Universal Robots PolyScope program: pourAndPutDown.urp

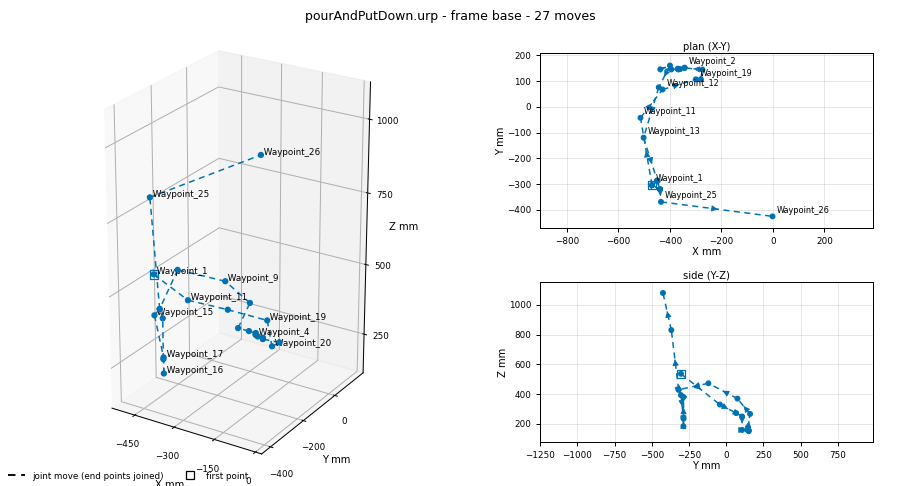
[picture p0: tool path of pourAndPutDown.urp in frame base, 27 of 27 moves have a stored position in this frame; points joined in program order, loops and branches not executed]
Program pourAndPutDown (installation=default directory=/programs/PrakjoyShi_Beer createdIn=5.12.6.1102099 lastSavedIn=5.12.6.1102099 robotSerialNumber=20215500597)
Calibrated DH parameters: a=[0.000193, -0.066673, -0.391568, -0.000012, 0.00005, 0]; d=[0.162643, -472.05677, 465.132521, 7.058239, 0.099746, 0.099582]; alpha=[1.571116, 0.00089, 0.003862, 1.569269, -1.569248, 0]; deltaTheta=[0, -1.413394, 7.628392, 0.068187, 0, -0.000001]
Robot Program (runOnlyOnce=true)
  MoveJ speed 60 deg/s, acceleration 80 deg/s^2 (useActiveTCP=true) feature=Base
    Waypoint Waypoint_1: TCP in base x=-469.422 y=-303.772 z=537.049 mm, rx=-0.9663 ry=-1.499 rz=1.6747 rad; joints [6.908, -106.662, 129.097, -206.194, -67.737, 6.591] deg; TCP offset x=0 y=0 z=191.5 mm, rx=0 ry=0 rz=0 rad
    Waypoint Waypoint_11: TCP in base x=-514.044 y=-42.229 z=330.478 mm, rx=0.9483 ry=1.8098 rz=-1.8406 rad; joints [-42.944, -57.453, 101.188, -230.29, 31.853, 49.611] deg
    Waypoint Waypoint_12: TCP in base x=-428.386 y=67.501 z=272.98 mm, rx=0.8234 ry=1.7173 rz=-1.638 rad; joints [-53.416, -47.466, 95.297, -230.558, 54.247, 53.558] deg
    Waypoint Waypoint_19: TCP in base x=-299.055 y=107.007 z=250.481 mm, rx=0.7818 ry=1.7818 rz=-1.7132 rad; joints [-69.052, -50.894, 107.804, -239.624, 68.324, 47.588] deg
    Waypoint Waypoint_20: TCP in base x=-279.734 y=106.984 z=159.803 mm, rx=0.7816 ry=1.7818 rz=-1.7132 rad; joints [-71.245, -40.233, 108.371, -250.83, 70.508, 47.507] deg
    Waypoint Waypoint_21: TCP in base x=-273.429 y=144.767 z=159.8 mm, rx=0.7817 ry=1.7819 rz=-1.7133 rad; joints [-73.337, -38.608, 103.329, -247.386, 72.596, 47.386] deg; TCP offset x=0 y=0 z=191.5 mm, rx=0 ry=0 rz=0 rad
    Waypoint Waypoint_2: TCP in base x=-342.426 y=151.266 z=151.388 mm, rx=0.9523 ry=1.6137 rz=-1.4653 rad; joints [-64.863, -34.688, 92.564, -242.174, 67.302, 65.082] deg; TCP offset x=0 y=0 z=191.5 mm, rx=0 ry=0 rz=0 rad
    Waypoint Waypoint_22: TCP in base x=-343.072 y=152.365 z=156.122 mm, rx=0.9896 ry=1.5509 rz=-1.4276 rad; joints [-64.858, -34.701, 92.594, -241.206, 67.284, 68.699] deg
    Waypoint Waypoint_3: TCP in base x=-360.092 y=146.777 z=158.442 mm, rx=1.1766 ry=1.3384 rz=-1.269 rad; joints [-64.056, -34.823, 92.755, -240.944, 64.321, 84.128] deg
    Wait Sleep waitTime=5
    Waypoint Waypoint_4: TCP in base x=-368.401 y=147.927 z=162.208 mm, rx=1.2276 ry=1.2595 rz=-1.2399 rad; joints [-64.055, -34.823, 92.749, -240.156, 62.793, 88.217] deg
    Wait Sleep waitTime=10
    Waypoint Waypoint_27: TCP in base x=-368.415 y=147.907 z=162.228 mm, rx=1.2493 ry=1.2256 rz=-1.2076 rad; joints [-64.053, -34.824, 92.753, -240.154, 62.79, 90.783] deg
    Wait Sleep waitTime=2
    Waypoint Waypoint_5: TCP in base x=-367.114 y=145.876 z=165.681 mm, rx=1.0874 ry=1.5479 rz=-1.4306 rad; joints [-64.058, -36.96, 92.743, -241.765, 62.844, 71.518] deg
    Waypoint Waypoint_6: TCP in base x=-367.053 y=145.733 z=170.165 mm, rx=0.9649 ry=1.707 rz=-1.5493 rad; joints [-64.058, -37.901, 92.741, -241.83, 62.842, 60.713] deg
    Waypoint Waypoint_7: TCP in base x=-394.155 y=145.769 z=170.181 mm, rx=0.9649 ry=1.707 rz=-1.5494 rad; joints [-61.586, -36.44, 89.13, -239.83, 60.388, 61.045] deg
    Waypoint Waypoint_8: TCP in base x=-437.191 y=145.775 z=170.185 mm, rx=0.9649 ry=1.707 rz=-1.5494 rad; joints [-57.925, -33.834, 82.842, -236.41, 56.767, 61.573] deg
    Waypoint Waypoint_10: TCP in base x=-399.525 y=160.604 z=267.522 mm, rx=0.291 ry=1.9476 rz=-1.9017 rad; joints [-57.921, -39.735, 82.866, -222.692, 65.755, 24.515] deg
    Waypoint Waypoint_9: TCP in base x=-443.299 y=75.819 z=370.314 mm, rx=-0.1462 ry=2.1698 rz=-2.071 rad; joints [-49.086, -50.8, 82.87, -214.951, 58.642, 3.159] deg
    Waypoint Waypoint_13: TCP in base x=-501.996 y=-119.391 z=473.346 mm, rx=-0.1865 ry=2.1452 rz=-2.0717 rad; joints [-29.839, -60.518, 82.876, -205.008, 41.125, 3.179] deg
    Waypoint Waypoint_14: TCP in base x=-438.339 y=-319.405 z=430.326 mm, rx=-0.0095 ry=-2.2019 rz=2.1503 rad; joints [-14.551, -76.261, 113.55, -222.987, 11.638, 3.16] deg
    Waypoint Waypoint_15: TCP in base x=-469.43 y=-303.759 z=393.841 mm, rx=-0.9664 ry=-1.499 rz=1.6746 rad; joints [6.93, -89.791, 142.194, -236.128, -67.835, 6.514] deg
    Waypoint Waypoint_17: TCP in base x=-447.918 y=-287.369 z=242.661 mm, rx=-0.8716 ry=-1.6291 rz=1.5246 rad; joints [1.903, -63.887, 152.292, -266.285, -61.848, -4.367] deg
    Waypoint Waypoint_16: TCP in base x=-447.928 y=-287.349 z=184.854 mm, rx=-0.8716 ry=-1.6291 rz=1.5245 rad; joints [1.931, -47.58, 150.654, -280.927, -61.868, -4.426] deg
    URCap Gripper (Robotiq_Grippers, Robotiq Inc.) dataModel(position=0.0, force=100.0, speed=100.0, positionInDouble=0.0, forceInDouble=100.0, speedInDouble=100.0, slaveIds=[9], blocking=true)
    Waypoint Waypoint_23: TCP in base x=-449.756 y=-286.313 z=235.635 mm, rx=-0.8887 ry=-1.6496 rz=1.5115 rad; joints [1.701, -63.9, 152.473, -264.905, -61.738, -4.834] deg
    Waypoint Waypoint_24: TCP in base x=-449.701 y=-286.338 z=380.979 mm, rx=-0.8887 ry=-1.6496 rz=1.5116 rad; joints [1.635, -100.122, 146.36, -222.64, -61.621, -4.69] deg
    Waypoint Waypoint_18: TCP in base x=-438.34 y=-319.404 z=430.315 mm, rx=-0.0095 ry=-2.2019 rz=2.1504 rad; joints [-14.551, -76.26, 113.551, -222.987, 11.638, 3.162] deg
    Waypoint Waypoint_25: TCP in base x=-434.434 y=-368.574 z=830.932 mm, rx=-0.0069 ry=-2.2054 rz=2.1858 rad; joints [-7.724, -82.704, 60.285, -160.607, 6.18, 1.676] deg
    Waypoint Waypoint_26: TCP in base x=-1.558 y=-424.817 z=1080.554 mm, rx=-0.0044 ry=-2.2185 rz=2.2204 rad; joints [-0.002, -89.999, -0.001, -89.999, 0.002, 0] deg
